Xinje XDPPro project, PLC1: XD5E-60T10 (software 3.5.3 2018-11-19)

PROGRAM Ladder

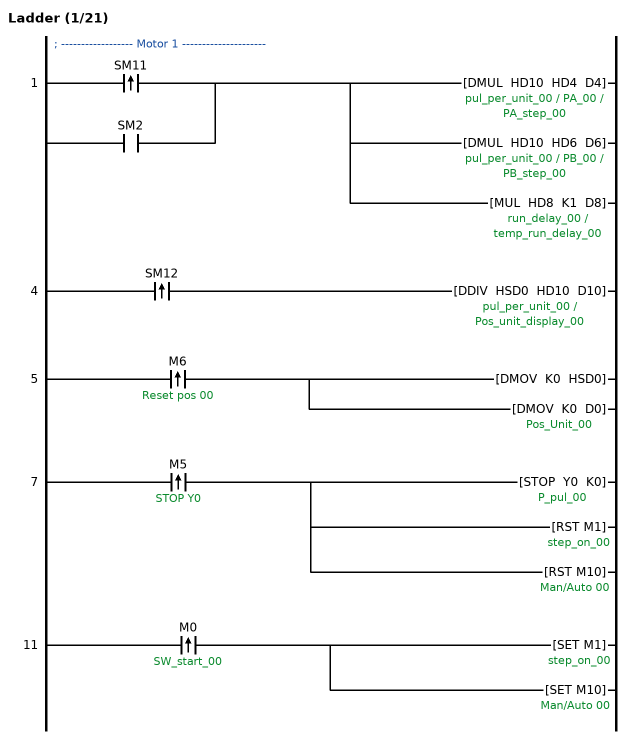
; ------------------ Motor 1 ---------------------
LDP    SM11
OR     SM2
DMUL   HD10 HD4 D4	; pul_per_unit_00 / PA_00 / PA_step_00
DMUL   HD10 HD6 D6	; pul_per_unit_00 / PB_00 / PB_step_00
MUL    HD8 K1 D8	; run_delay_00 / temp_run_delay_00
LDP    SM12
DDIV   HSD0 HD10 D10	; pul_per_unit_00 / Pos_unit_display_00
LDP    M6	; Reset pos 00
DMOV   K0 HSD0
DMOV   K0 D0	; Pos_Unit_00
LDP    M5	; STOP Y0
STOP   Y0 K0	; P_pul_00
RST    M1	; step_on_00
RST    M10	; Man/Auto 00
LDP    M0	; SW_start_00
SET    M1	; step_on_00
SET    M10	; Man/Auto 00

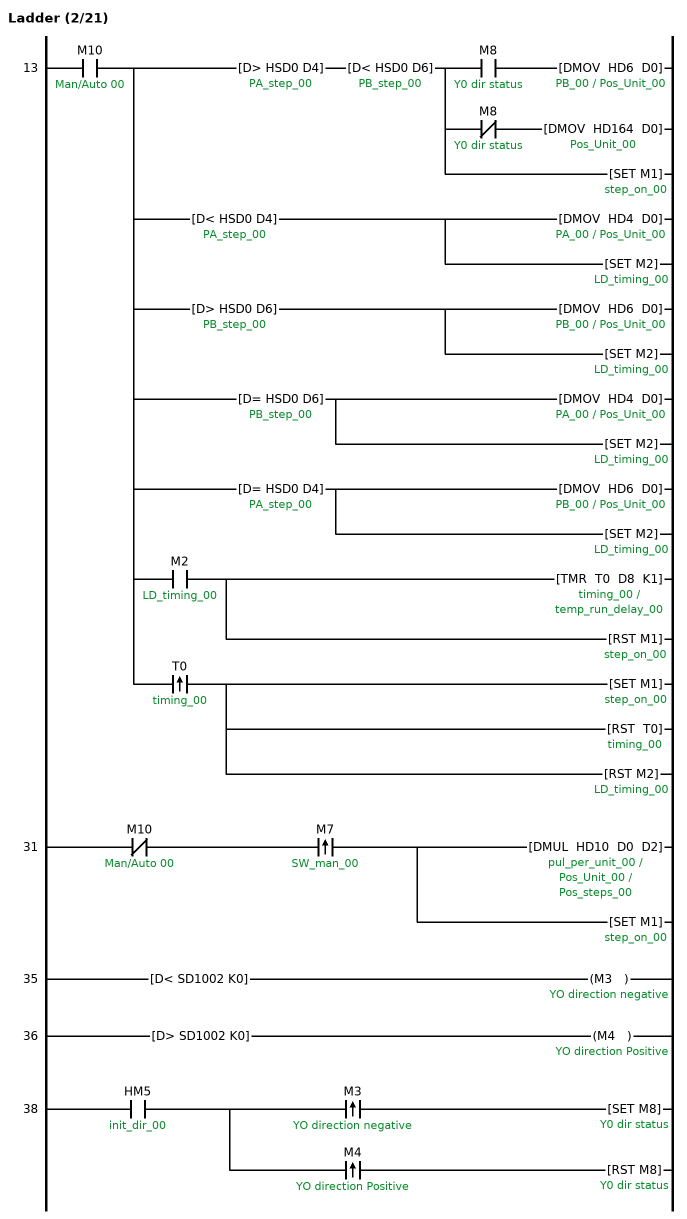
LD     M10	; Man/Auto 00
MPS
DAND>  HSD0 D4	; PA_step_00
DAND<  HSD0 D6	; PB_step_00
MPS
AND    M8	; Y0 dir status
DMOV   HD6 D0	; PB_00 / Pos_Unit_00
MRD
ANI    M8	; Y0 dir status
DMOV   HD164 D0	; Pos_Unit_00
MPP
SET    M1	; step_on_00
MRD
DAND<  HSD0 D4	; PA_step_00
DMOV   HD4 D0	; PA_00 / Pos_Unit_00
SET    M2	; LD_timing_00
MRD
DAND>  HSD0 D6	; PB_step_00
DMOV   HD6 D0	; PB_00 / Pos_Unit_00
SET    M2	; LD_timing_00
MRD
DAND=  HSD0 D6	; PB_step_00
DMOV   HD4 D0	; PA_00 / Pos_Unit_00
SET    M2	; LD_timing_00
MRD
DAND=  HSD0 D4	; PA_step_00
DMOV   HD6 D0	; PB_00 / Pos_Unit_00
SET    M2	; LD_timing_00
MRD
AND    M2	; LD_timing_00
TMR    T0 D8 K1	; timing_00 / temp_run_delay_00
RST    M1	; step_on_00
MPP
ANDP   T0	; timing_00
SET    M1	; step_on_00
RST    T0	; timing_00
RST    M2	; LD_timing_00
LDI    M10	; Man/Auto 00
ANDP   M7	; SW_man_00
DMUL   HD10 D0 D2	; pul_per_unit_00 / Pos_Unit_00 / Pos_steps_00
SET    M1	; step_on_00
DLD<   SD1002 K0
OUT    M3	; YO direction negative
DLD>   SD1002 K0
OUT    M4	; YO direction Positive
LD     HM5	; init_dir_00
MPS
ANDP   M3	; YO direction negative
SET    M8	; Y0 dir status
MPP
ANDP   M4	; YO direction Positive
RST    M8	; Y0 dir status

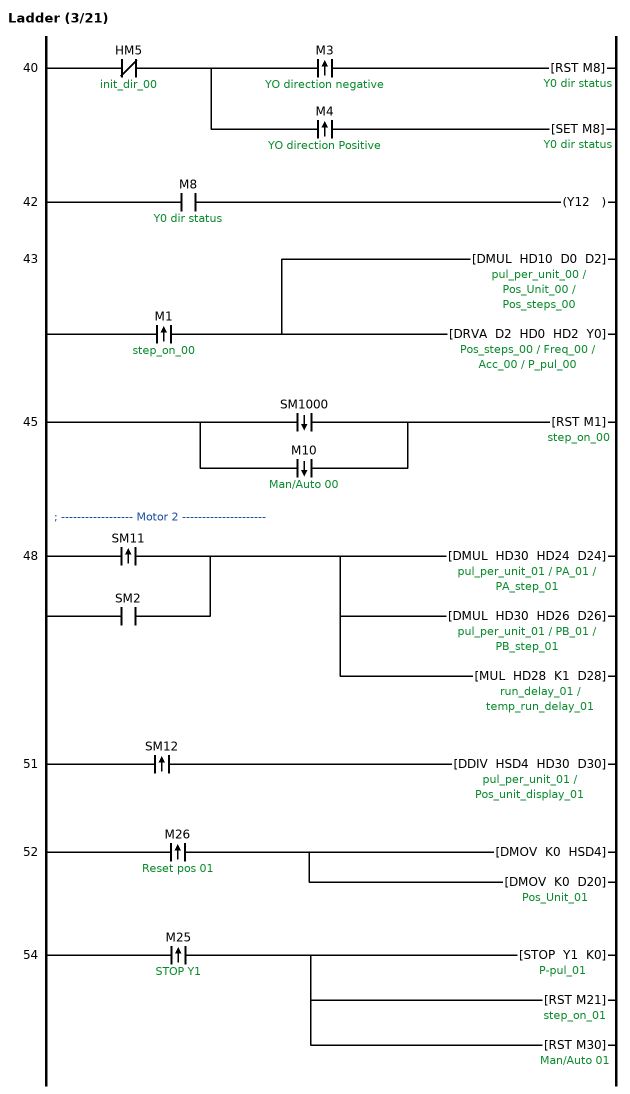
LDI    HM5	; init_dir_00
MPS
ANDP   M3	; YO direction negative
RST    M8	; Y0 dir status
MPP
ANDP   M4	; YO direction Positive
SET    M8	; Y0 dir status
LD     M8	; Y0 dir status
OUT    Y12
LDP    M1	; step_on_00
DMUL   HD10 D0 D2	; pul_per_unit_00 / Pos_Unit_00 / Pos_steps_00
DRVA   D2 HD0 HD2 Y0	; Pos_steps_00 / Freq_00 / Acc_00 / P_pul_00
LDF    SM1000
ORF    M10	; Man/Auto 00
RST    M1	; step_on_00
; ------------------ Motor 2 ---------------------
LDP    SM11
OR     SM2
DMUL   HD30 HD24 D24	; pul_per_unit_01 / PA_01 / PA_step_01
DMUL   HD30 HD26 D26	; pul_per_unit_01 / PB_01 / PB_step_01
MUL    HD28 K1 D28	; run_delay_01 / temp_run_delay_01
LDP    SM12
DDIV   HSD4 HD30 D30	; pul_per_unit_01 / Pos_unit_display_01
LDP    M26	; Reset pos 01
DMOV   K0 HSD4
DMOV   K0 D20	; Pos_Unit_01
LDP    M25	; STOP Y1
STOP   Y1 K0	; P-pul_01
RST    M21	; step_on_01
RST    M30	; Man/Auto 01

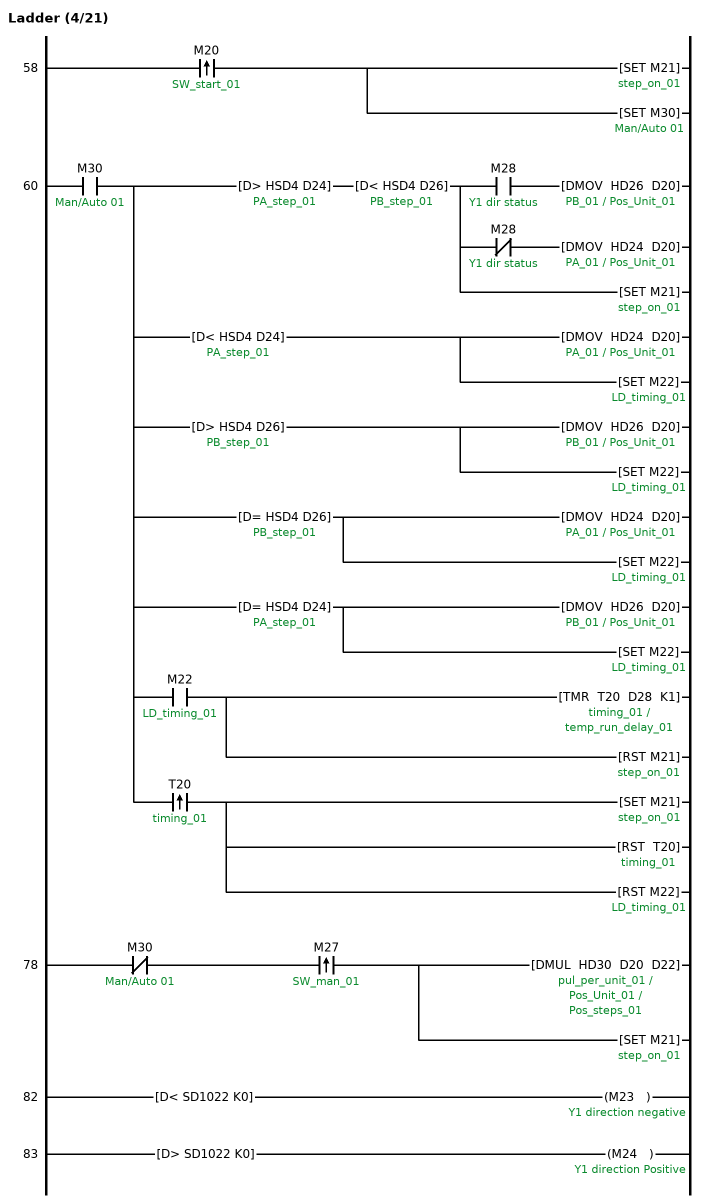
LDP    M20	; SW_start_01
SET    M21	; step_on_01
SET    M30	; Man/Auto 01
LD     M30	; Man/Auto 01
MPS
DAND>  HSD4 D24	; PA_step_01
DAND<  HSD4 D26	; PB_step_01
MPS
AND    M28	; Y1 dir status
DMOV   HD26 D20	; PB_01 / Pos_Unit_01
MRD
ANI    M28	; Y1 dir status
DMOV   HD24 D20	; PA_01 / Pos_Unit_01
MPP
SET    M21	; step_on_01
MRD
DAND<  HSD4 D24	; PA_step_01
DMOV   HD24 D20	; PA_01 / Pos_Unit_01
SET    M22	; LD_timing_01
MRD
DAND>  HSD4 D26	; PB_step_01
DMOV   HD26 D20	; PB_01 / Pos_Unit_01
SET    M22	; LD_timing_01
MRD
DAND=  HSD4 D26	; PB_step_01
DMOV   HD24 D20	; PA_01 / Pos_Unit_01
SET    M22	; LD_timing_01
MRD
DAND=  HSD4 D24	; PA_step_01
DMOV   HD26 D20	; PB_01 / Pos_Unit_01
SET    M22	; LD_timing_01
MRD
AND    M22	; LD_timing_01
TMR    T20 D28 K1	; timing_01 / temp_run_delay_01
RST    M21	; step_on_01
MPP
ANDP   T20	; timing_01
SET    M21	; step_on_01
RST    T20	; timing_01
RST    M22	; LD_timing_01
LDI    M30	; Man/Auto 01
ANDP   M27	; SW_man_01
DMUL   HD30 D20 D22	; pul_per_unit_01 / Pos_Unit_01 / Pos_steps_01
SET    M21	; step_on_01
DLD<   SD1022 K0
OUT    M23	; Y1 direction negative
DLD>   SD1022 K0
OUT    M24	; Y1 direction Positive

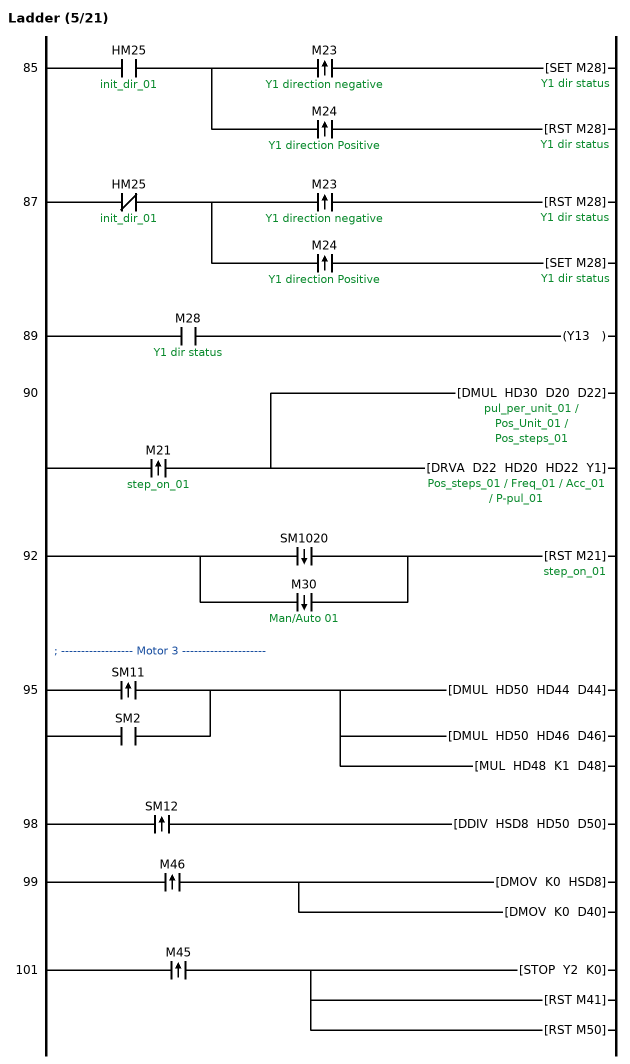
LD     HM25	; init_dir_01
MPS
ANDP   M23	; Y1 direction negative
SET    M28	; Y1 dir status
MPP
ANDP   M24	; Y1 direction Positive
RST    M28	; Y1 dir status
LDI    HM25	; init_dir_01
MPS
ANDP   M23	; Y1 direction negative
RST    M28	; Y1 dir status
MPP
ANDP   M24	; Y1 direction Positive
SET    M28	; Y1 dir status
LD     M28	; Y1 dir status
OUT    Y13
LDP    M21	; step_on_01
DMUL   HD30 D20 D22	; pul_per_unit_01 / Pos_Unit_01 / Pos_steps_01
DRVA   D22 HD20 HD22 Y1	; Pos_steps_01 / Freq_01 / Acc_01 / P-pul_01
LDF    SM1020
ORF    M30	; Man/Auto 01
RST    M21	; step_on_01
; ------------------ Motor 3 ---------------------
LDP    SM11
OR     SM2
DMUL   HD50 HD44 D44
DMUL   HD50 HD46 D46
MUL    HD48 K1 D48
LDP    SM12
DDIV   HSD8 HD50 D50
LDP    M46
DMOV   K0 HSD8
DMOV   K0 D40
LDP    M45
STOP   Y2 K0
RST    M41
RST    M50

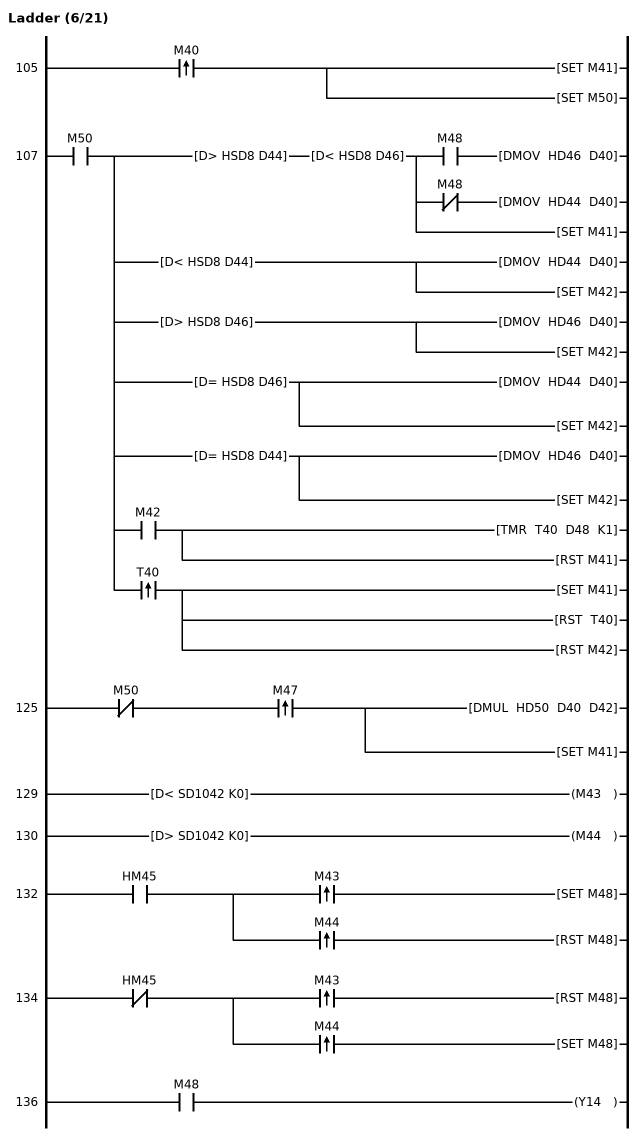
LDP    M40
SET    M41
SET    M50
LD     M50
MPS
DAND>  HSD8 D44
DAND<  HSD8 D46
MPS
AND    M48
DMOV   HD46 D40
MRD
ANI    M48
DMOV   HD44 D40
MPP
SET    M41
MRD
DAND<  HSD8 D44
DMOV   HD44 D40
SET    M42
MRD
DAND>  HSD8 D46
DMOV   HD46 D40
SET    M42
MRD
DAND=  HSD8 D46
DMOV   HD44 D40
SET    M42
MRD
DAND=  HSD8 D44
DMOV   HD46 D40
SET    M42
MRD
AND    M42
TMR    T40 D48 K1
RST    M41
MPP
ANDP   T40
SET    M41
RST    T40
RST    M42
LDI    M50
ANDP   M47
DMUL   HD50 D40 D42
SET    M41
DLD<   SD1042 K0
OUT    M43
DLD>   SD1042 K0
OUT    M44
LD     HM45
MPS
ANDP   M43
SET    M48
MPP
ANDP   M44
RST    M48
LDI    HM45
MPS
ANDP   M43
RST    M48
MPP
ANDP   M44
SET    M48
LD     M48
OUT    Y14

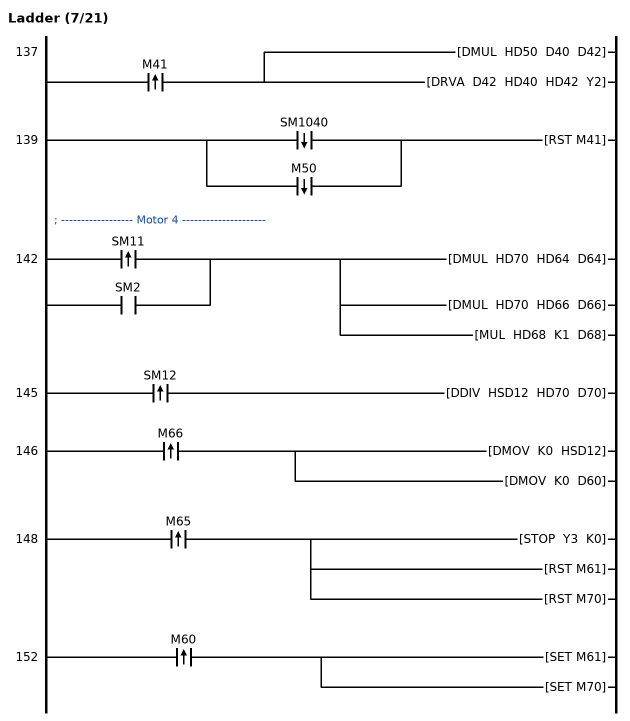
LDP    M41
DMUL   HD50 D40 D42
DRVA   D42 HD40 HD42 Y2
LDF    SM1040
ORF    M50
RST    M41
; ------------------ Motor 4 ---------------------
LDP    SM11
OR     SM2
DMUL   HD70 HD64 D64
DMUL   HD70 HD66 D66
MUL    HD68 K1 D68
LDP    SM12
DDIV   HSD12 HD70 D70
LDP    M66
DMOV   K0 HSD12
DMOV   K0 D60
LDP    M65
STOP   Y3 K0
RST    M61
RST    M70
LDP    M60
SET    M61
SET    M70

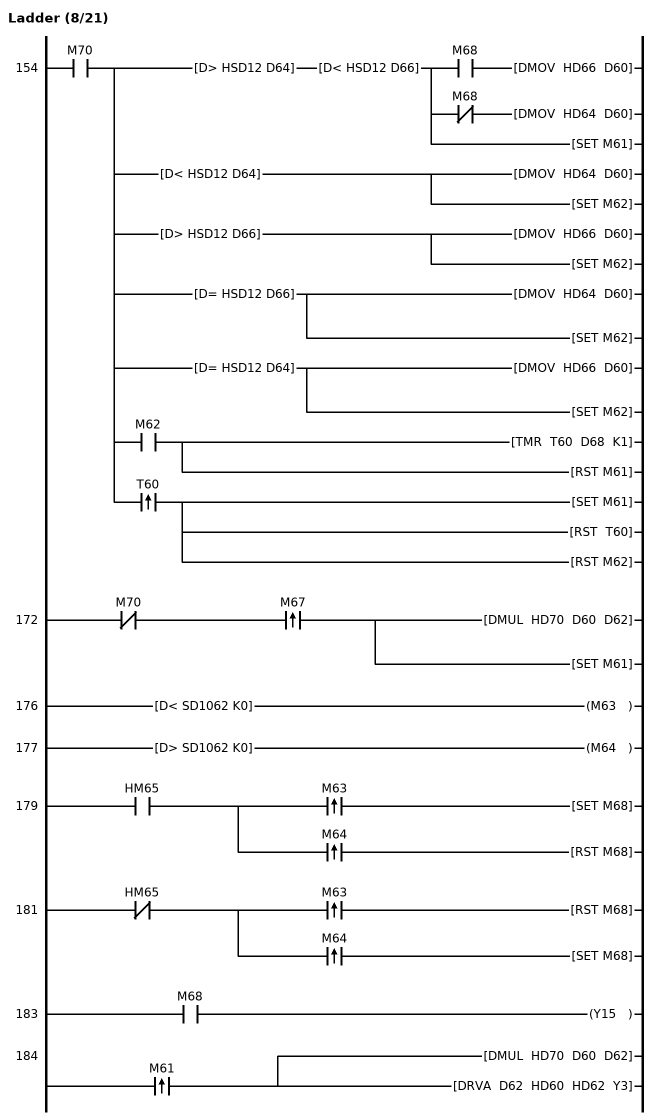
LD     M70
MPS
DAND>  HSD12 D64
DAND<  HSD12 D66
MPS
AND    M68
DMOV   HD66 D60
MRD
ANI    M68
DMOV   HD64 D60
MPP
SET    M61
MRD
DAND<  HSD12 D64
DMOV   HD64 D60
SET    M62
MRD
DAND>  HSD12 D66
DMOV   HD66 D60
SET    M62
MRD
DAND=  HSD12 D66
DMOV   HD64 D60
SET    M62
MRD
DAND=  HSD12 D64
DMOV   HD66 D60
SET    M62
MRD
AND    M62
TMR    T60 D68 K1
RST    M61
MPP
ANDP   T60
SET    M61
RST    T60
RST    M62
LDI    M70
ANDP   M67
DMUL   HD70 D60 D62
SET    M61
DLD<   SD1062 K0
OUT    M63
DLD>   SD1062 K0
OUT    M64
LD     HM65
MPS
ANDP   M63
SET    M68
MPP
ANDP   M64
RST    M68
LDI    HM65
MPS
ANDP   M63
RST    M68
MPP
ANDP   M64
SET    M68
LD     M68
OUT    Y15
LDP    M61
DMUL   HD70 D60 D62
DRVA   D62 HD60 HD62 Y3

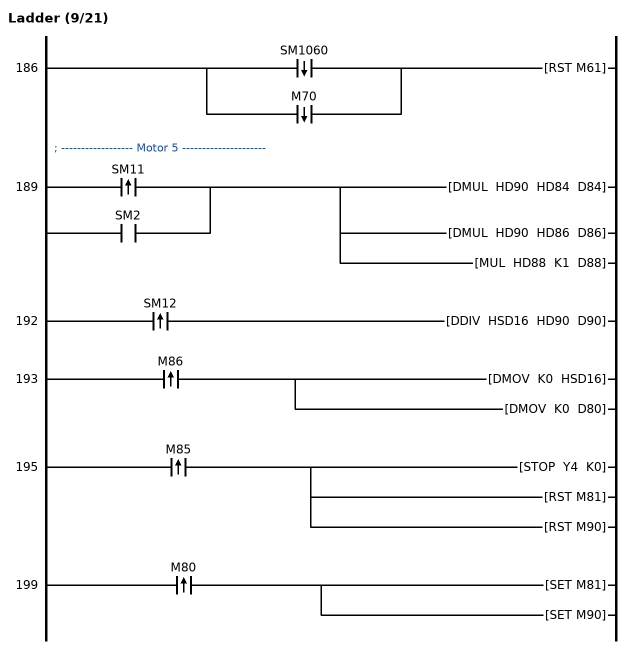
LDF    SM1060
ORF    M70
RST    M61
; ------------------ Motor 5 ---------------------
LDP    SM11
OR     SM2
DMUL   HD90 HD84 D84
DMUL   HD90 HD86 D86
MUL    HD88 K1 D88
LDP    SM12
DDIV   HSD16 HD90 D90
LDP    M86
DMOV   K0 HSD16
DMOV   K0 D80
LDP    M85
STOP   Y4 K0
RST    M81
RST    M90
LDP    M80
SET    M81
SET    M90

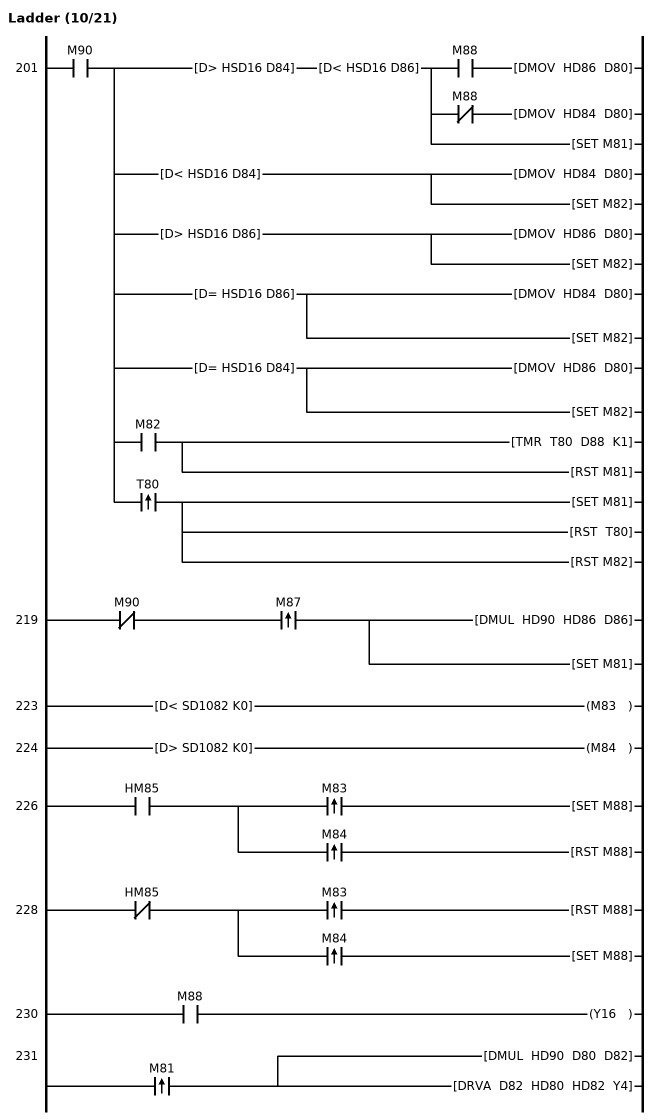
LD     M90
MPS
DAND>  HSD16 D84
DAND<  HSD16 D86
MPS
AND    M88
DMOV   HD86 D80
MRD
ANI    M88
DMOV   HD84 D80
MPP
SET    M81
MRD
DAND<  HSD16 D84
DMOV   HD84 D80
SET    M82
MRD
DAND>  HSD16 D86
DMOV   HD86 D80
SET    M82
MRD
DAND=  HSD16 D86
DMOV   HD84 D80
SET    M82
MRD
DAND=  HSD16 D84
DMOV   HD86 D80
SET    M82
MRD
AND    M82
TMR    T80 D88 K1
RST    M81
MPP
ANDP   T80
SET    M81
RST    T80
RST    M82
LDI    M90
ANDP   M87
DMUL   HD90 HD86 D86
SET    M81
DLD<   SD1082 K0
OUT    M83
DLD>   SD1082 K0
OUT    M84
LD     HM85
MPS
ANDP   M83
SET    M88
MPP
ANDP   M84
RST    M88
LDI    HM85
MPS
ANDP   M83
RST    M88
MPP
ANDP   M84
SET    M88
LD     M88
OUT    Y16
LDP    M81
DMUL   HD90 D80 D82
DRVA   D82 HD80 HD82 Y4

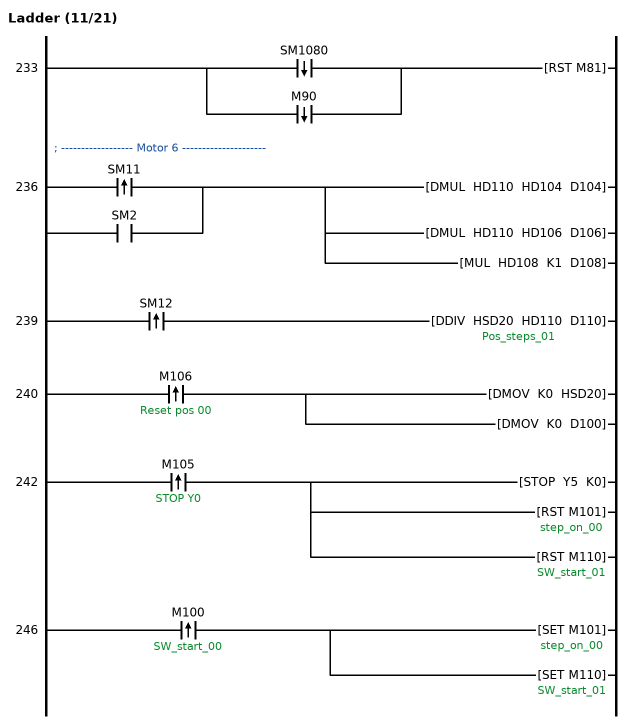
LDF    SM1080
ORF    M90
RST    M81
; ------------------ Motor 6 ---------------------
LDP    SM11
OR     SM2
DMUL   HD110 HD104 D104
DMUL   HD110 HD106 D106
MUL    HD108 K1 D108
LDP    SM12
DDIV   HSD20 HD110 D110	; Pos_steps_01
LDP    M106	; Reset pos 00
DMOV   K0 HSD20
DMOV   K0 D100
LDP    M105	; STOP Y0
STOP   Y5 K0
RST    M101	; step_on_00
RST    M110	; SW_start_01
LDP    M100	; SW_start_00
SET    M101	; step_on_00
SET    M110	; SW_start_01

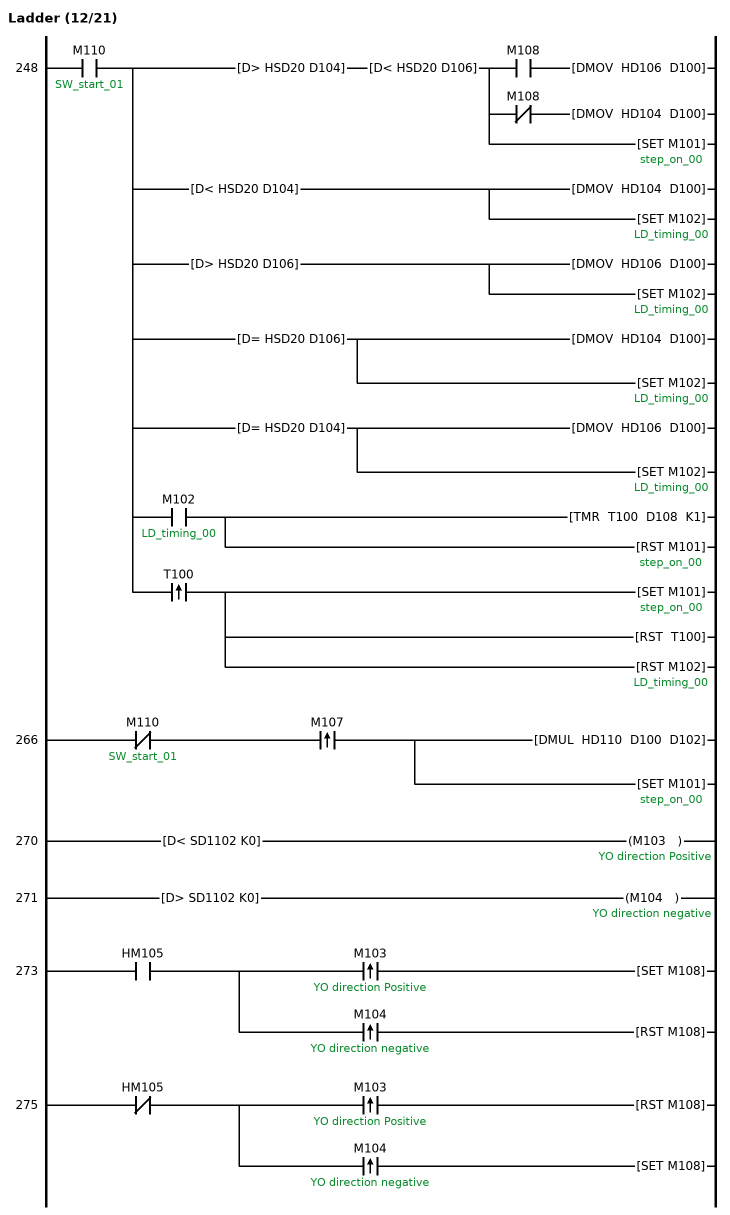
LD     M110	; SW_start_01
MPS
DAND>  HSD20 D104
DAND<  HSD20 D106
MPS
AND    M108
DMOV   HD106 D100
MRD
ANI    M108
DMOV   HD104 D100
MPP
SET    M101	; step_on_00
MRD
DAND<  HSD20 D104
DMOV   HD104 D100
SET    M102	; LD_timing_00
MRD
DAND>  HSD20 D106
DMOV   HD106 D100
SET    M102	; LD_timing_00
MRD
DAND=  HSD20 D106
DMOV   HD104 D100
SET    M102	; LD_timing_00
MRD
DAND=  HSD20 D104
DMOV   HD106 D100
SET    M102	; LD_timing_00
MRD
AND    M102	; LD_timing_00
TMR    T100 D108 K1
RST    M101	; step_on_00
MPP
ANDP   T100
SET    M101	; step_on_00
RST    T100
RST    M102	; LD_timing_00
LDI    M110	; SW_start_01
ANDP   M107
DMUL   HD110 D100 D102
SET    M101	; step_on_00
DLD<   SD1102 K0
OUT    M103	; YO direction Positive
DLD>   SD1102 K0
OUT    M104	; YO direction negative
LD     HM105
MPS
ANDP   M103	; YO direction Positive
SET    M108
MPP
ANDP   M104	; YO direction negative
RST    M108
LDI    HM105
MPS
ANDP   M103	; YO direction Positive
RST    M108
MPP
ANDP   M104	; YO direction negative
SET    M108

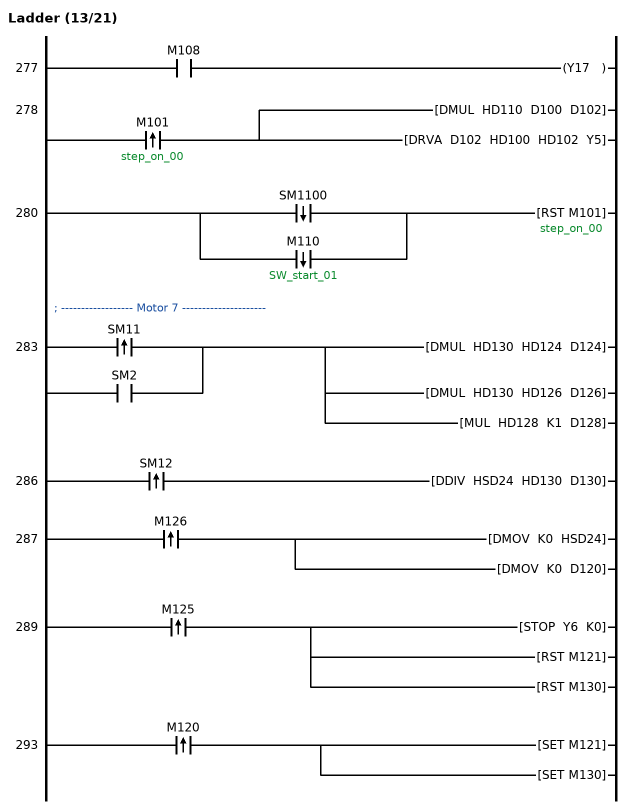
LD     M108
OUT    Y17
LDP    M101	; step_on_00
DMUL   HD110 D100 D102
DRVA   D102 HD100 HD102 Y5
LDF    SM1100
ORF    M110	; SW_start_01
RST    M101	; step_on_00
; ------------------ Motor 7 ---------------------
LDP    SM11
OR     SM2
DMUL   HD130 HD124 D124
DMUL   HD130 HD126 D126
MUL    HD128 K1 D128
LDP    SM12
DDIV   HSD24 HD130 D130
LDP    M126
DMOV   K0 HSD24
DMOV   K0 D120
LDP    M125
STOP   Y6 K0
RST    M121
RST    M130
LDP    M120
SET    M121
SET    M130

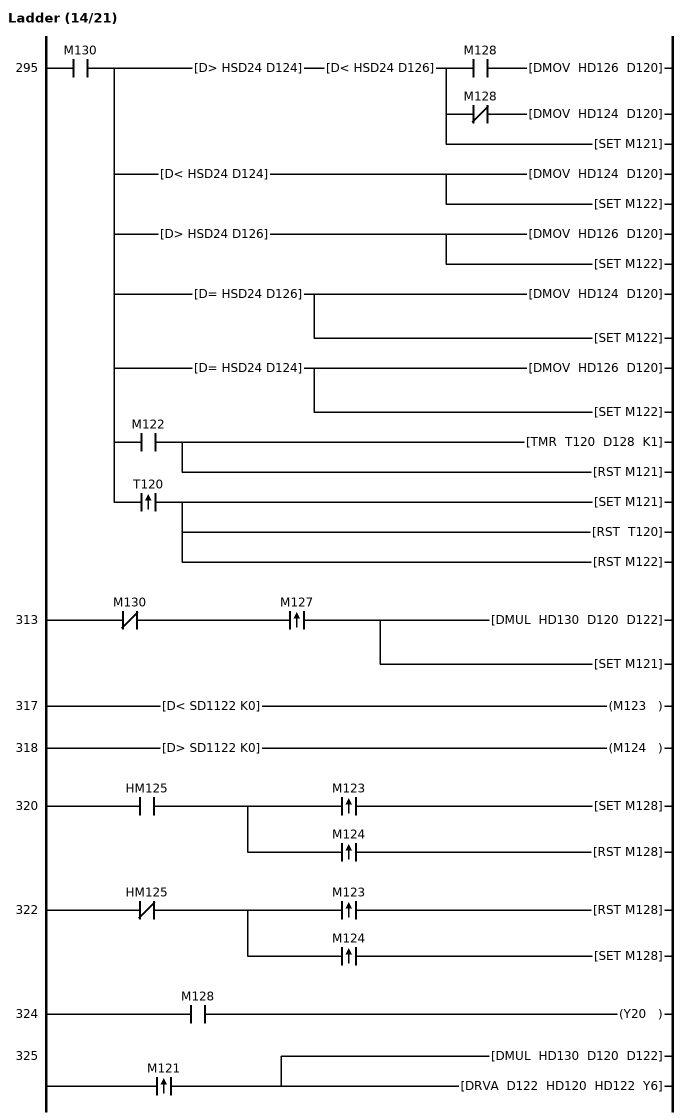
LD     M130
MPS
DAND>  HSD24 D124
DAND<  HSD24 D126
MPS
AND    M128
DMOV   HD126 D120
MRD
ANI    M128
DMOV   HD124 D120
MPP
SET    M121
MRD
DAND<  HSD24 D124
DMOV   HD124 D120
SET    M122
MRD
DAND>  HSD24 D126
DMOV   HD126 D120
SET    M122
MRD
DAND=  HSD24 D126
DMOV   HD124 D120
SET    M122
MRD
DAND=  HSD24 D124
DMOV   HD126 D120
SET    M122
MRD
AND    M122
TMR    T120 D128 K1
RST    M121
MPP
ANDP   T120
SET    M121
RST    T120
RST    M122
LDI    M130
ANDP   M127
DMUL   HD130 D120 D122
SET    M121
DLD<   SD1122 K0
OUT    M123
DLD>   SD1122 K0
OUT    M124
LD     HM125
MPS
ANDP   M123
SET    M128
MPP
ANDP   M124
RST    M128
LDI    HM125
MPS
ANDP   M123
RST    M128
MPP
ANDP   M124
SET    M128
LD     M128
OUT    Y20
LDP    M121
DMUL   HD130 D120 D122
DRVA   D122 HD120 HD122 Y6

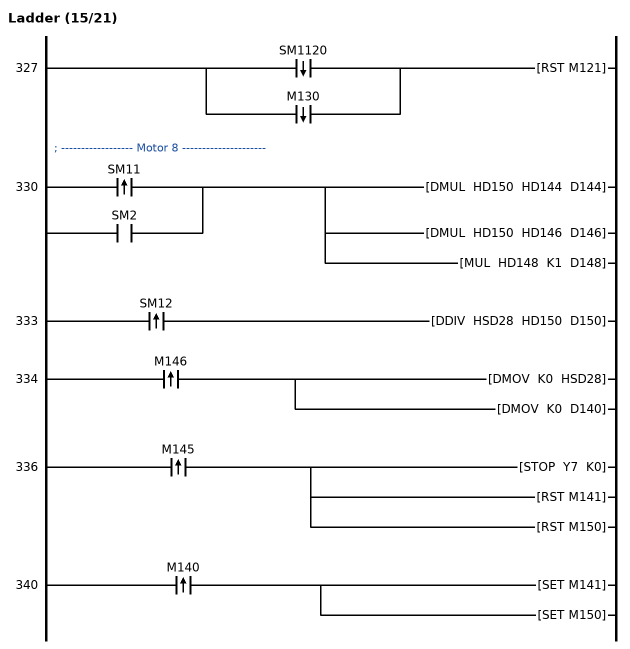
LDF    SM1120
ORF    M130
RST    M121
; ------------------ Motor 8 ---------------------
LDP    SM11
OR     SM2
DMUL   HD150 HD144 D144
DMUL   HD150 HD146 D146
MUL    HD148 K1 D148
LDP    SM12
DDIV   HSD28 HD150 D150
LDP    M146
DMOV   K0 HSD28
DMOV   K0 D140
LDP    M145
STOP   Y7 K0
RST    M141
RST    M150
LDP    M140
SET    M141
SET    M150

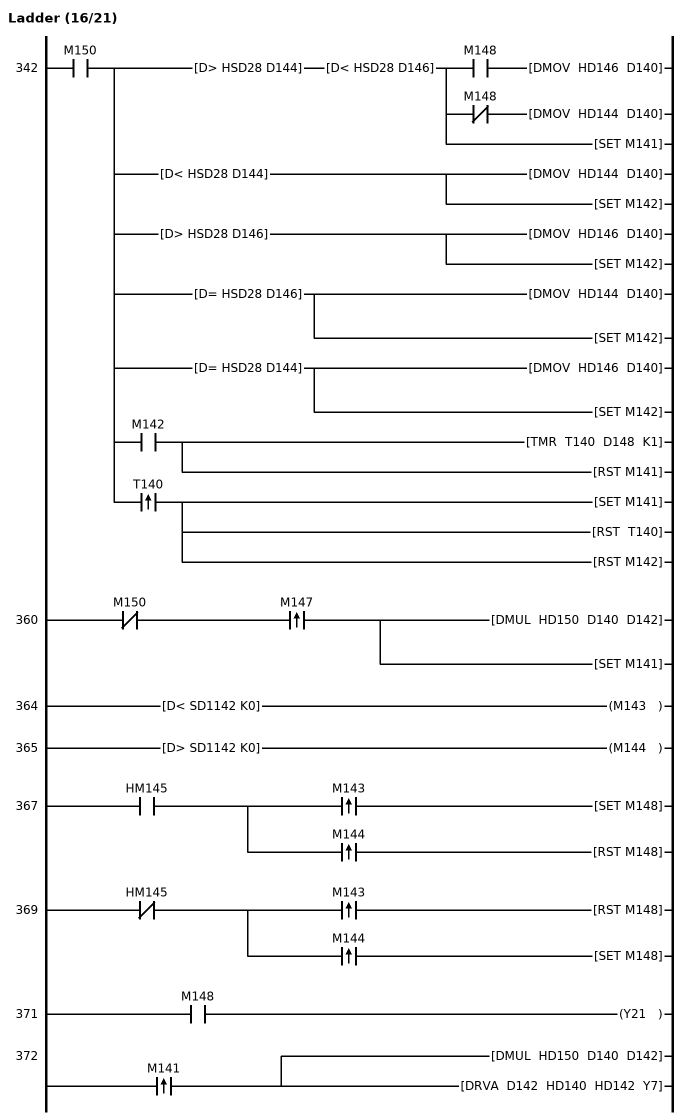
LD     M150
MPS
DAND>  HSD28 D144
DAND<  HSD28 D146
MPS
AND    M148
DMOV   HD146 D140
MRD
ANI    M148
DMOV   HD144 D140
MPP
SET    M141
MRD
DAND<  HSD28 D144
DMOV   HD144 D140
SET    M142
MRD
DAND>  HSD28 D146
DMOV   HD146 D140
SET    M142
MRD
DAND=  HSD28 D146
DMOV   HD144 D140
SET    M142
MRD
DAND=  HSD28 D144
DMOV   HD146 D140
SET    M142
MRD
AND    M142
TMR    T140 D148 K1
RST    M141
MPP
ANDP   T140
SET    M141
RST    T140
RST    M142
LDI    M150
ANDP   M147
DMUL   HD150 D140 D142
SET    M141
DLD<   SD1142 K0
OUT    M143
DLD>   SD1142 K0
OUT    M144
LD     HM145
MPS
ANDP   M143
SET    M148
MPP
ANDP   M144
RST    M148
LDI    HM145
MPS
ANDP   M143
RST    M148
MPP
ANDP   M144
SET    M148
LD     M148
OUT    Y21
LDP    M141
DMUL   HD150 D140 D142
DRVA   D142 HD140 HD142 Y7

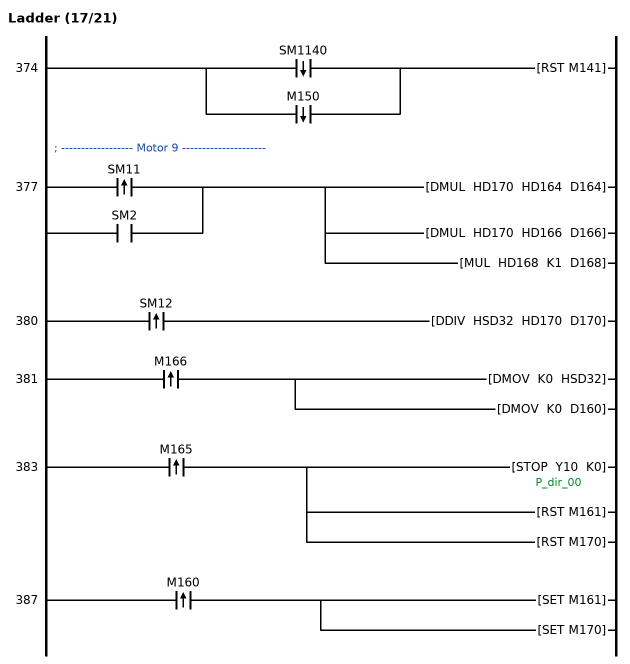
LDF    SM1140
ORF    M150
RST    M141
; ------------------ Motor 9 ---------------------
LDP    SM11
OR     SM2
DMUL   HD170 HD164 D164
DMUL   HD170 HD166 D166
MUL    HD168 K1 D168
LDP    SM12
DDIV   HSD32 HD170 D170
LDP    M166
DMOV   K0 HSD32
DMOV   K0 D160
LDP    M165
STOP   Y10 K0	; P_dir_00
RST    M161
RST    M170
LDP    M160
SET    M161
SET    M170

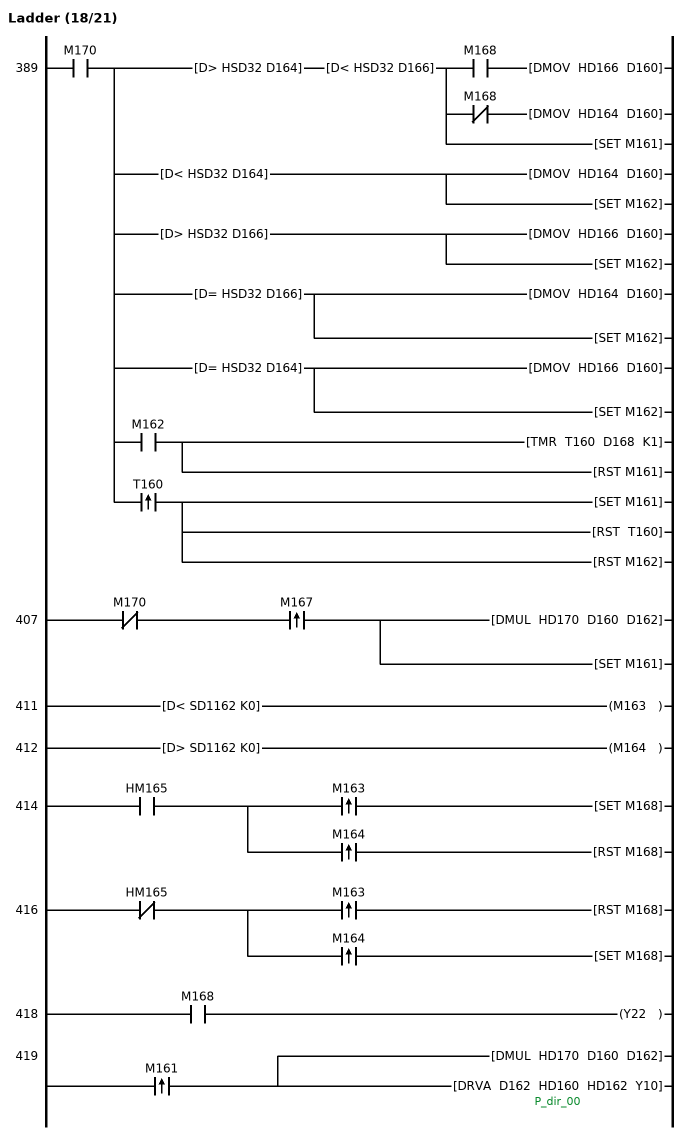
LD     M170
MPS
DAND>  HSD32 D164
DAND<  HSD32 D166
MPS
AND    M168
DMOV   HD166 D160
MRD
ANI    M168
DMOV   HD164 D160
MPP
SET    M161
MRD
DAND<  HSD32 D164
DMOV   HD164 D160
SET    M162
MRD
DAND>  HSD32 D166
DMOV   HD166 D160
SET    M162
MRD
DAND=  HSD32 D166
DMOV   HD164 D160
SET    M162
MRD
DAND=  HSD32 D164
DMOV   HD166 D160
SET    M162
MRD
AND    M162
TMR    T160 D168 K1
RST    M161
MPP
ANDP   T160
SET    M161
RST    T160
RST    M162
LDI    M170
ANDP   M167
DMUL   HD170 D160 D162
SET    M161
DLD<   SD1162 K0
OUT    M163
DLD>   SD1162 K0
OUT    M164
LD     HM165
MPS
ANDP   M163
SET    M168
MPP
ANDP   M164
RST    M168
LDI    HM165
MPS
ANDP   M163
RST    M168
MPP
ANDP   M164
SET    M168
LD     M168
OUT    Y22
LDP    M161
DMUL   HD170 D160 D162
DRVA   D162 HD160 HD162 Y10	; P_dir_00

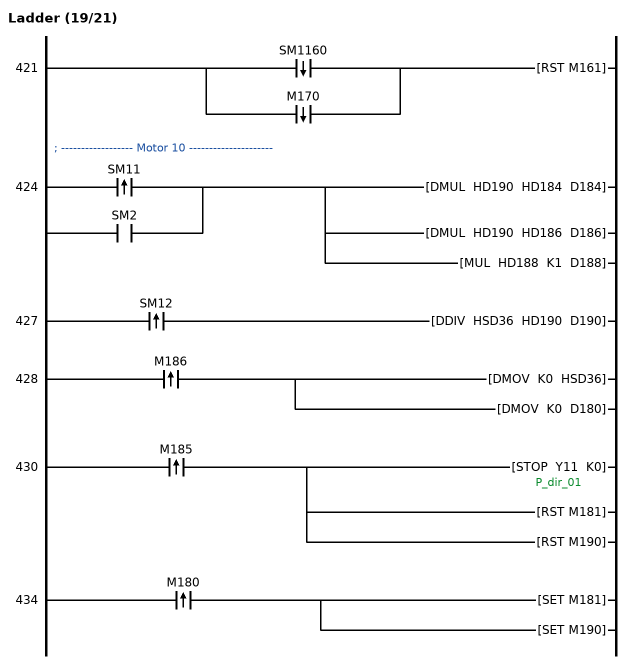
LDF    SM1160
ORF    M170
RST    M161
; ------------------ Motor 10 ---------------------
LDP    SM11
OR     SM2
DMUL   HD190 HD184 D184
DMUL   HD190 HD186 D186
MUL    HD188 K1 D188
LDP    SM12
DDIV   HSD36 HD190 D190
LDP    M186
DMOV   K0 HSD36
DMOV   K0 D180
LDP    M185
STOP   Y11 K0	; P_dir_01
RST    M181
RST    M190
LDP    M180
SET    M181
SET    M190

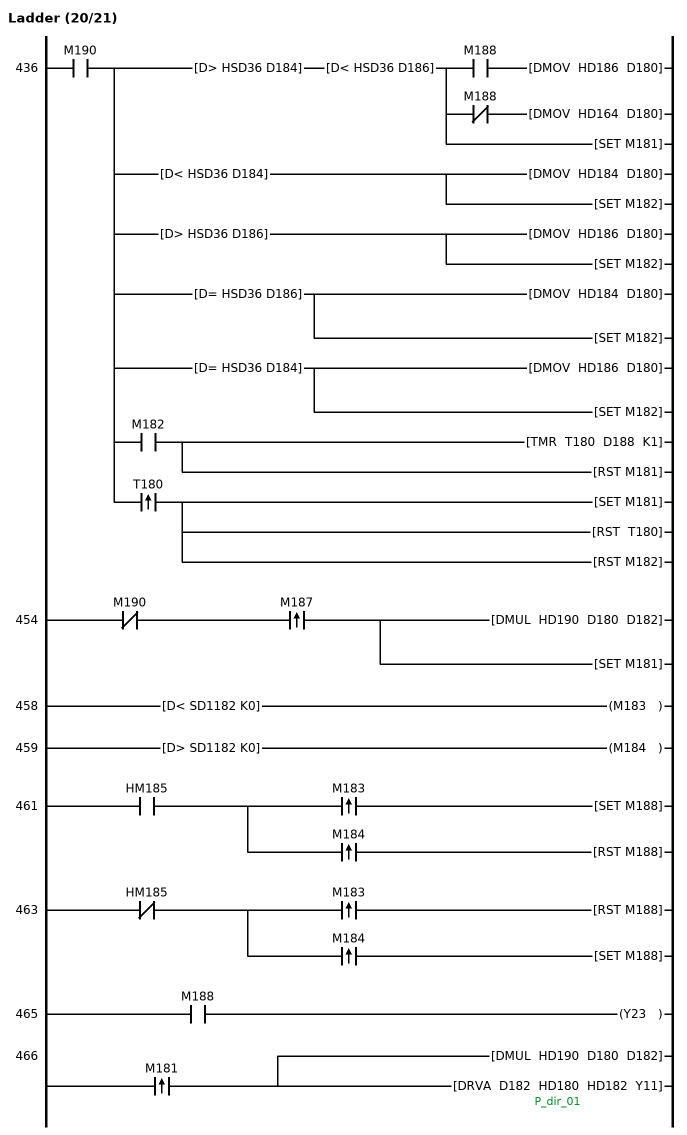
LD     M190
MPS
DAND>  HSD36 D184
DAND<  HSD36 D186
MPS
AND    M188
DMOV   HD186 D180
MRD
ANI    M188
DMOV   HD164 D180
MPP
SET    M181
MRD
DAND<  HSD36 D184
DMOV   HD184 D180
SET    M182
MRD
DAND>  HSD36 D186
DMOV   HD186 D180
SET    M182
MRD
DAND=  HSD36 D186
DMOV   HD184 D180
SET    M182
MRD
DAND=  HSD36 D184
DMOV   HD186 D180
SET    M182
MRD
AND    M182
TMR    T180 D188 K1
RST    M181
MPP
ANDP   T180
SET    M181
RST    T180
RST    M182
LDI    M190
ANDP   M187
DMUL   HD190 D180 D182
SET    M181
DLD<   SD1182 K0
OUT    M183
DLD>   SD1182 K0
OUT    M184
LD     HM185
MPS
ANDP   M183
SET    M188
MPP
ANDP   M184
RST    M188
LDI    HM185
MPS
ANDP   M183
RST    M188
MPP
ANDP   M184
SET    M188
LD     M188
OUT    Y23
LDP    M181
DMUL   HD190 D180 D182
DRVA   D182 HD180 HD182 Y11	; P_dir_01

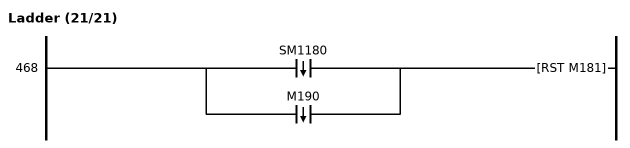
LDF    SM1180
ORF    M190
RST    M181

COMMENTS (devices not used above)
D202	Pos 01
D204	Tan so 01
D206	Gia toc 01
HD200	Step_per_unit_00